{attribute 'linkalways'} 
{attribute 'no_explicit_call' := 'This FB is a CLASS and must be accessed using methods or properties'}
{attribute 'enable_dynamic_creation'}
FUNCTION_BLOCK Node_RGBA_GREEN EXTENDS VisionNode
VAR
    out : _TcVnVector4_LREAL;
END_VAR

METHOD PUBLIC  Clone : I_Node
VAR
	pNode : POINTER TO Node_RGBA_GREEN;
END_VAR
pNode := __NEW(Node_RGBA_GREEN);
Clone := pNode^;
END_METHOD

METHOD FB_init : BOOL
VAR_INPUT
	bInitRetains : BOOL; // if TRUE, the retain variables are initialized (warm start / cold start)
	bInCopyCode : BOOL;  // if TRUE, the instance afterwards gets moved into the copy code (online change)
END_VAR
AddOutput('out', out);
END_METHOD

METHOD PROTECTED OnExecute : HRESULT
out.Value := GVL_COLOURS.RGBA_GREEN;
END_METHOD

METHOD PUBLIC PreExecutionCheck
VAR_INPUT
	Check : I_PreExecutionChecks;
END_VAR
END_METHOD

END_FUNCTION_BLOCK

(* stored: Version 1.1.0.1, ProductVersion 3.1.4024.13
   POU Node_RGBA_GREEN: Id {4226ff1c-08c2-077e-1b03-83b20b3a19b7}, SpecialFunc None
   Folder Constructor: Id {2cf7b7f2-45c3-081b-0e85-008b38c9121f}
   Method Clone: Id {c1e91962-a5ad-0dfc-1846-d969feac632f}
   Method FB_init: Id {b2280364-84dc-09ab-25d8-f808dd2a0eef}
   Method OnExecute: Id {4148d0f4-ef24-09dd-34f6-40389dade783}
   Method PreExecutionCheck: Id {f76241cf-9243-0f5e-1e44-bbd96d0ad1e7} *)
